{attribute 'conditionalshow'}
FUNCTION_BLOCK FB_KNXMaster_Messages
VAR_INPUT
	{attribute 'hide'}
	bErrorKNX							: BOOL;						//Error from the Mbus Function
	{attribute 'hide'}
	bErrorIntern						: BOOL;						//Internal Error
	{attribute 'hide'}
	bWarning							: BOOL;						//Warning from the RTU Function
	{attribute 'hide'}
	iWarningCode						: INT;						//Warning Code
	{attribute 'hide'}
	iErrorCode							: INT;						//Error Code		
END_VAR
VAR_OUTPUT
	{attribute 'hide'}
	byErrorWarning						: BYTE;						//Error Warning State
	eMessageKNXMaster					: E_Message_KNXMaster;		//Message from the KNX Master Function
END_VAR
VAR
END_VAR

//Creator : Kai Ebensperger
//Company : Lynus AG
//Date : 24.08.2021
//Version : 1.0.0.0

//With this Funciton is possible to handel the Error and Warning Codes from the KNX Master.

//Warnings
IF bWarning AND iWarningCode = 0 THEN
	eMessageKNXMaster := E_Message_KNXMaster.eNoConnectionToBackend;
END_IF

//Intern Errors
IF bErrorIntern AND iErrorCode = 1 THEN
	eMessageKNXMaster := E_Message_KNXMaster.eTooMuchKNXMasters;
END_IF
//KNX Errors
IF bErrorKNX AND iErrorCode = 1 THEN
	eMessageKNXMaster := E_Message_KNXMaster.eWrong_KNX_Phys_Addr;
ELSIF bErrorKNX AND iErrorCode = 2 THEN
	eMessageKNXMaster := E_Message_KNXMaster.eWrong_KNX_Group_Addr;
ELSIF bErrorKNX AND iErrorCode = 3 THEN
	eMessageKNXMaster := E_Message_KNXMaster.eWrong_KNX_Group_Len;
ELSIF bErrorKNX AND iErrorCode = 4 THEN
	eMessageKNXMaster := E_Message_KNXMaster.eWrong_KNX_No_Filter;
ELSIF bErrorKNX AND iErrorCode = 10 THEN
	eMessageKNXMaster := E_Message_KNXMaster.eWrong_KNX_Firmware;
ELSIF bErrorKNX AND iErrorCode = 11 THEN
	eMessageKNXMaster := E_Message_KNXMaster.eWrong_KNX_Mode;
ELSIF bErrorKNX AND iErrorCode = 12 THEN
	eMessageKNXMaster := E_Message_KNXMaster.eWrong_Mode;
ELSIF bErrorKNX AND iErrorCode = 14 THEN
	eMessageKNXMaster := E_Message_KNXMaster.eWrong_KNX_Firmware_B1_Necessary;
ELSIF bErrorKNX AND iErrorCode = 15 THEN
	eMessageKNXMaster := E_Message_KNXMaster.eWrong_KNX_Firmware_B3_Necessary;
ELSIF bErrorKNX AND iErrorCode = 20 THEN
	eMessageKNXMaster := E_Message_KNXMaster.eWrong_KNX_Data_Len;
ELSIF bErrorKNX AND iErrorCode = 21 THEN
	eMessageKNXMaster := E_Message_KNXMaster.eError_KNX_Service_Not_Support;
ELSIF bErrorKNX AND iErrorCode = 30 THEN
	eMessageKNXMaster := E_Message_KNXMaster.eKL6301_TP_Toggle_Error;
ELSIF bErrorKNX AND iErrorCode = 31 THEN
	eMessageKNXMaster := E_Message_KNXMaster.eTime_Out;
ELSIF bErrorKNX AND iErrorCode = 32 THEN
	eMessageKNXMaster := E_Message_KNXMaster.eKL6301_No_Response_from_Terminal;
ELSIF bErrorKNX AND iErrorCode = 40 THEN
	eMessageKNXMaster := E_Message_KNXMaster.eError_Send_8Bit_Wrong_Scaling_Mode;
ELSIF bErrorKNX AND iErrorCode = 100 THEN
	eMessageKNXMaster := E_Message_KNXMaster.eError_KNX_Phy_Addr_Not_Support;
ELSIF bErrorKNX AND iErrorCode = 101 THEN
	eMessageKNXMaster := E_Message_KNXMaster.eError_KNX_Write_Data;
ELSIF bErrorKNX AND iErrorCode = 102 THEN
	eMessageKNXMaster := E_Message_KNXMaster.eMonitor_Mode_Len_Is_Not_Ok_Must_0;
ELSIF bErrorKNX AND iErrorCode = 103 THEN
	eMessageKNXMaster := E_Message_KNXMaster.eMonitor_Mode_Addr_Is_Not_Ok_Must_0;
ELSIF bErrorKNX AND iErrorCode = 104 THEN
	eMessageKNXMaster := E_Message_KNXMaster.eWatchdog_Error_No_Send;
ELSIF bErrorKNX AND iErrorCode = 16#0BBB THEN
	eMessageKNXMaster := E_Message_KNXMaster.eError_KNX_No_Ack;
ELSIF bErrorKNX AND iErrorCode = 16#FAFB THEN
	eMessageKNXMaster := E_Message_KNXMaster.eError_KNX_No_Com_To_TP;
ELSIF bErrorKNX AND iErrorCode = 16#0FCC THEN
	eMessageKNXMaster := E_Message_KNXMaster.eError_TP_Temp_Warning;
ELSIF bErrorKNX AND iErrorCode = 16#17CC THEN
	eMessageKNXMaster := E_Message_KNXMaster.eError_TP_Protocol_Error;
ELSIF bErrorKNX AND iErrorCode = 16#27CC THEN
	eMessageKNXMaster := E_Message_KNXMaster.eError_TP_Transmitter_Error;
ELSIF bErrorKNX AND iErrorCode = 16#47CC THEN
	eMessageKNXMaster := E_Message_KNXMaster.eError_TP_Receive_Error;
ELSIF bErrorKNX AND iErrorCode = 16#87CC THEN
	eMessageKNXMaster := E_Message_KNXMaster.eError_TP_Slave_Collision;
END_IF 

IF bWarning THEN 
	byErrorWarning := 1;
END_IF	
	IF bErrorKNX OR bErrorIntern THEN
		byErrorWarning := 2;
	END_IF

//All ok
IF NOT bErrorKNX AND NOT bErrorIntern AND NOT bWarning THEN
	eMessageKNXMaster := E_Message_KNXMaster.eAllOk;
		byErrorWarning := 0;
END_IF

END_FUNCTION_BLOCK

(* stored: Version 1.1.0.1, ProductVersion 3.1.4024.9
   POU FB_KNXMaster_Messages: Id {90e2af8f-b020-42c6-be60-056a507644db}, SpecialFunc None *)
